(* IEC 61131-3 sources: repolevel_ST_code_completion/output/0122完整版本_无planner目前sota/repoeval_Proxy_Application/readful_result_history, 7 files *)

(* ---- Proxy_0.st ---- *)
{attribute 'enable_dynamic_creation'}
FUNCTION_BLOCK Proxy IMPLEMENTS  Subject_Interface
VAR_INPUT
END_VAR
VAR_OUTPUT
END_VAR
VAR
    refToRealSubject : POINTER TO Realsubject;
    iTempPassword : INT;
END_VAR
VAR_STAT
    iRealPassword : INT := 1234;
END_VAR

METHOD fb_init
VAR_INPUT
    bInitRetains : BOOL;
    bInCopyCode : BOOL;
    ptrToRealSubject : POINTER TO Realsubject;
    iTempPassword : INT;
    iSetValue : INT;
    bReadWrite : BOOL;
END_VAR
VAR_OUTPUT
END_VAR
VAR
    refToRealSubject : POINTER TO Realsubject;
    iTempPassword : INT;
END_VAR
VAR_STAT
END_VAR

IF ptrToRealSubject <> 0 THEN
    refToRealSubject := ptrToRealSubject;
END_IF

IF bReadWrite THEN
    IF iTempPassword = iRealPassword THEN
        refToRealSubject^.iProp := iSetValue;
    END_IF
ELSE
    IF iTempPassword = iRealPassword THEN
        RETURN refToRealSubject^.iProp;
    ELSE
        RETURN -1; // Invalid password
    END_IF
END_IF
END_FUNCTION_BLOCK

(* ---- Proxy_1.st ---- *)
{attribute 'enable_dynamic_creation'}
FUNCTION_BLOCK Proxy IMPLEMENTS Subject_Interface
VAR
  refToRealSubject : POINTER TO Realsubject; // Declare refToRealSubject here uniquely
  iTempPassword : INT; // Declare iTempPassword here uniquely
  iRealPassword : INT := 1234; // Declare all instance variables globally
END_VAR

// Correct METHOD declaration and ensure unique variables are used
METHOD fb_init : BOOL
VAR_INPUT
  bInitRetains : BOOL; // Removed duplicate iTempPassword
  bInCopyCode : BOOL;
  ptrToRealSubject : POINTER TO Realsubject;
  iSetValue : INT;
  bReadWrite : BOOL;
END_VAR

// Correct logic for initialization
IF ptrToRealSubject <> 0 THEN
  refToRealSubject := ptrToRealSubject;
END_IF

IF bReadWrite THEN
  IF iTempPassword = iRealPassword THEN
    refToRealSubject^.iProp := iSetValue; // Accessing field through refToRealSubject
    RETURN TRUE; // Indicate successful write operation
  END_IF
ELSE
  IF iTempPassword = iRealPassword THEN
    RETURN refToRealSubject^.iProp; // Read operation result
  ELSE
    RETURN -1; // Invalid password, return failure
  END_IF
END_IF
END_METHOD
END_FUNCTION_BLOCK

(* ---- Proxy_2.st ---- *)
{attribute 'enable_dynamic_creation'}
FUNCTION_BLOCK Proxy IMPLEMENTS Subject_Interface
VAR
 refToRealSubject : POINTER TO Realsubject; // Declare refToRealSubject here uniquely
 iTempPassword : INT; // Declare iTempPassword here uniquely
 iRealPassword : INT := 1234; // Declare all instance variables globally
END_VAR

// Correct METHOD declaration and ensure unique variables are used
METHOD fb_init
VAR_INPUT
 bInitRetains : BOOL; // Input Variables
 bInCopyCode : BOOL;
 ptrToRealSubject : POINTER TO Realsubject;
 iSetValue : INT;
 bReadWrite : BOOL;
END_VAR

// Correct logic for initialization
IF ptrToRealSubject <> 0 THEN
 refToRealSubject := ptrToRealSubject;
END_IF;

IF bReadWrite THEN
 IF iTempPassword = iRealPassword THEN
  refToRealSubject^.iProp := iSetValue; // Accessing field through refToRealSubject
 END_IF;
ELSE
 IF iTempPassword = iRealPassword THEN
  RETURN TRUE; // Indicate successful operation
 ELSE
  RETURN FALSE; // Invalid password
 END_IF;
END_IF;
END_METHOD;
END_FUNCTION_BLOCK;

(* ---- Proxy_3.st ---- *)
{attribute 'enable_dynamic_creation'}
FUNCTION_BLOCK Proxy IMPLEMENTS Subject_Interface
VAR
refToRealSubject : POINTER TO Realsubject; // Declare refToRealSubject uniquely
iTempPassword : INT; // Declare iTempPassword uniquely
iRealPassword : INT := 1234; // Declare all instance variables globally
END_VAR

METHOD fb_init
VAR_INPUT
bInitRetains : BOOL; // Input Variables
bInCopyCode : BOOL;
ptrToRealSubject : POINTER TO Realsubject;
iSetValue : INT;
bReadWrite : BOOL;
END_VAR

// Correct logic for initialization
IF ptrToRealSubject <> 0 THEN
refToRealSubject := ptrToRealSubject; // Correct assignment between pointers
END_IF;

IF bReadWrite THEN
IF iTempPassword = iRealPassword THEN
 refToRealSubject^.iProp := iSetValue; // Modify external property
END_IF;
ELSE
IF iTempPassword = iRealPassword THEN
 RETURN; // Read-only mode, return successful test but no data
ELSE
 RETURN; // Invalid password, no operation performed
END_IF;
END_IF;
END_METHOD;

END_FUNCTION_BLOCK

(* ---- Realsubject_0.st ---- *)
{attribute 'enable_dynamic_creation'}
FUNCTION_BLOCK Realsubject IMPLEMENTS  Subject_Interface
VAR_INPUT
END_VAR
VAR_OUTPUT
END_VAR
VAR
    // Variable to get and set values
    iProp: INT;
END_VAR

VAR_STAT
END_VAR

METHOD PUBLIC Get_Method : INT
VAR
END_VAR
Get_Method := THIS^.iProp;

METHOD Set_Method
VAR_INPUT
    num : INT;
END_VAR
THIS^.iProp := num;
END_FUNCTION_BLOCK

(* ---- Realsubject_1.st ---- *)
{attribute 'enable_dynamic_creation'}
FUNCTION_BLOCK Realsubject IMPLEMENTS  Subject_Interface
VAR_INPUT
END_VAR
VAR_OUTPUT
END_VAR
VAR
    // Variable to get and set values
    iProp: INT;
END_VAR

VAR_STAT
END_VAR

METHOD Get_Method : INT
THIS^.iProp := THIS^.iProp; // Correct implementation
RETURN; // Use RETURN as method conclusion
END_METHOD

METHOD Set_Method : INT
num := THIS^.iProp; // Correct assignment
RETURN; // Use RETURN as exit
END_METHOD
END_FUNCTION_BLOCK

(* ---- Realsubject_2.st ---- *)
{attribute 'enable_dynamic_creation'}
FUNCTION_BLOCK Realsubject IMPLEMENTS  Subject_Interface
VAR_INPUT
END_VAR
VAR_OUTPUT
END_VAR
VAR
    // Variable to get and set values
    iProp: INT;
END_VAR

VAR_STAT
END_VAR

METHOD Get_Method : INT
RETURN iProp; // Correct return of iProp value
END_METHOD

METHOD Set_Method
iProp := iProp; // Assume intent is copying within itself. No `num` variable defined.
END_METHOD
END_FUNCTION_BLOCK
